(* IEC 61131-3 sources: BODAS-HelloWorld/extracted_st/bodas_rc18_12_40/plc_logic/application/02_easyconfig/easyconfig_import/bds_in_ec/bds_in_ec_gvl, 1 file *)

(* ---- bds_in_ec_gvl.st ---- *)
(* --- Interface --- *)
{attribute 'qualified_only' := ''}
VAR_GLOBAL CONSTANT
    BDS_inCmn_postVariants_DU8 : USINT := 1;
END_VAR
